FUNCTION_BLOCK FB_RemoteControl
VAR_INPUT
END_VAR
VAR_OUTPUT
END_VAR
VAR
	itfCommand		: I_Command;
END_VAR

METHOD pressButton : BOOL
VAR_INPUT
END_VAR
itfCommand.execute();
END_METHOD

METHOD setCommand : BOOL
VAR_INPUT
	command		:I_Command;
END_VAR
itfCommand := command;
END_METHOD

END_FUNCTION_BLOCK

(* stored: Version 1.1.0.1
   POU FB_RemoteControl: Id {0fffc3b9-fe55-4ebb-bbc3-e01e7f08edb6}, SpecialFunc None
   Method pressButton: Id {f0edecf8-a039-40d8-aa69-8ef55080de41}
   Method setCommand: Id {5d4c0292-797a-4526-9ab2-5dbaac6da562} *)
